FUNCTION_BLOCK RunUnitIndexerMaster EXTENDS RunUnitTransporterBase
VAR		
	Axis : POINTER TO RunAxis; //axis reference
	
	//Working registers
	nCounter : DINT;
	
	
END_VAR
VAR PERSISTENT
END_VAR

SUPER^(); // call base class's execution

//---------------
//	S16#0-S16#0F : regular state as standard indexer
//	S16#10 : mechanical control of movement
//---------------

CASE outputState OF
	16#0:
		//-------------------------
		//	Trigger all slaves
		//-------------------------
		FOR nCounter:=1 TO 3 BY 1 DO
			slaveWorkingSignal[nCounter] := slaveLinkageStatus[nCounter];
		END_FOR
		bSerialTransition := TRUE;
	16#1:	
		//------------------------------------------
		//check material synchronization to Databse
		//All slot act must be off
		//------------------------------------------
		bSerialTransition := TRUE;
		FOR nCounter:=0 TO SlotCount-1 BY 1 DO
			bSerialTransition := bSerialTransition AND NOT SlotBase[nCounter].Act;
		END_FOR
	16#2:
		//--------------------------------
		// Scanning working signal until all are off
		//--------------------------------
		bSerialTransition := TRUE;
		FOR nCounter:= 1 TO 32 BY 1 DO
			bSerialTransition := bSerialTransition AND NOT slaveWorkingSignal[nCounter];
		END_FOR
	16#3:
		//-------------------
		//Sync with down stream
		//-------------------
		IF syncEngaged AND syncAcknowledged THEN
			syncEngaged := FALSE; //reset
		END_IF
		bSerialTransition := NOT syncAcknowledged; //make sure signal is resetted
		IF bSerialTransition THEN
			//move last slot's information to buffer area
			syncMatId:= SlotLast^.Id; // for the last slot
			syncMatValid := SlotLast^.Valid;// ready to sync
		END_IF
	16#4:
		//2 modes
		// a. synchronize with downstream only, go with pull upstream if avialable
		// b. synchronize with down/upstream both
	
		// pull by downstream (set on then check off
		// pull upstream (check on then reset
		
		IF syncMatValid AND NOT syncEngaged THEN
			syncEngaged := TRUE;//ready to synchronizing (communicate with downstream
		END_IF
		
		//listen to move
		bSerialTransition :=  (NOT syncMatValid) OR (syncAcknowledged AND syncMatValid);
		IF bSerialTransition THEN
			NextState := 16#10;
		END_IF
	16#10:
		//---------------------
		//shifting movement mechaincal
		//---------------------	
	16#F:
		//---------------------------------------------------------------
		//Do data shifting (move is valid/id) , leave first slot as empty
		//---------------------------------------------------------------
		FOR nCounter:=SlotCount-1 TO 0 BY -1 DO
			IF nCounter > 0 THEN
				SlotBase[nCounter].Id := SlotBase[nCounter-1].id;
				SlotBase[nCounter].Valid := SlotBase[nCounter-1].Valid;
			END_IF			
		END_FOR
		bSerialTransition := TRUE;	
END_CASE

METHOD FB_init : BOOL
VAR_INPUT
	bInitRetains : BOOL; // if TRUE, the retain variables are initialized (warm start / cold start)
	bInCopyCode : BOOL;  // if TRUE, the instance afterwards gets moved into the copy code (online change)
	
	argParent : POINTER TO RunUnitGeneric;
	argSlotBase : POINTER TO RunMaterial;
	argSlotLast : POINTER TO RunMaterial;
	
	argUpstream : POINTER TO RunUnitTransporterBase;
	argAxis : POINTER TO RunAxis;

END_VAR
//initialize 
Parent := argParent;
SlotBase := argSlotBase;
SlotLast := argSlotLast;

Axis := argAxis;
Upstream := argUpstream;

IF Upstream=0 THEN
	isProxyMode:=TRUE; //no upstream , i am proxy
END_IF

//calculate how much slot related
SlotCount :=  TO_INT((SlotLast-SlotBase)/SIZEOF(RunMaterial) + 1);
END_METHOD

END_FUNCTION_BLOCK

(* stored: Version 1.1.0.1, ProductVersion 3.1.4024.0
   POU RunUnitIndexerMaster: Id {2551b589-75e5-432e-8b87-41fecbcdc1e1}, SpecialFunc None
   Method FB_init: Id {b6ef164b-1316-42c1-8dbc-2d2d314e57b5} *)
